(* CODESYS project SmartTraffic.project

Project tree, tasks and I/O mapping:
  Device : CODESYS Control Win V3, 3S - Smart Software Solutions GmbH, order no. 305021, version 3.5.5.50
    application Application
      libraries: Standard, * (System); MQTT Client Library, 3.5.13.20 (Stefan Roßmann Engineering Solutions)
      task MainTask (cyclic, interval t#20ms, priority 1) calls PLC_PRG
      task VISU_TASK (cyclic, interval 100 ms, priority 31) calls VisuElems.Visu_Prg
      program PLC_PRG [CFC]
      function block TrafficLight [ST]
      visualisation Visualization
  text list GlobalTextList
*)

// Device/Application/PLC_PRG
PROGRAM PLC_PRG
VAR
	MQTT_Client_FB_MQTTClient_1 : MQTT_Client.FB_MQTTClient;
	TrafficLight_1: TrafficLight;
END_VAR

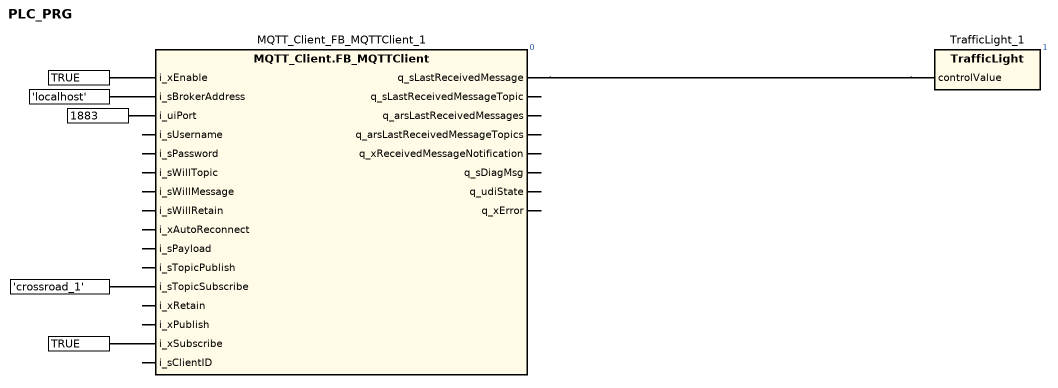
MQTT_Client_FB_MQTTClient_1(
    i_xEnable := TRUE,
    i_sBrokerAddress := 'localhost',
    i_uiPort := 1883,
    i_sTopicSubscribe := 'crossroad_1',
    i_xSubscribe := TRUE); // MQTT_Client.FB_MQTTClient
TrafficLight_1(controlValue := MQTT_Client_FB_MQTTClient_1.q_sLastReceivedMessage); // TrafficLight

END_PROGRAM

// Device/Application/TrafficLight
FUNCTION_BLOCK TrafficLight
VAR_INPUT
	controlValue: STRING;
END_VAR
VAR_OUTPUT
END_VAR
VAR
	Street1Red:BOOL;
	Street1Green:BOOL;
	Street2Red:BOOL;
	Street2Green:BOOL;
	Amber:BOOL;
	Street_TON_1:TON;
	Street_TON_2:TON;
	controlValue_TON_3:TON;
	lastControlValue: STRING;
	street1: TIME := T#15S;
	street2: TIME := T#15S;
	CTU_1: CTU;
	R_TRIG_1: R_TRIG;
END_VAR

CTU_1(PV:= 1, CU:= controlValue_TON_3.Q);
IF CTU_1.Q THEN 
	IF controlValue = 'Increase' THEN 
		street1:= street1 + T#10S;
		street2:= street2 - T#10S;
	ELSIF controlValue = 'Lower' THEN 
		street1:= street1 - T#10S;
		street2:= street2 + T#10S;
	END_IF
	CTU_1(RESET:= TRUE);
	CTU_1(RESET:= FALSE);
	controlValue_TON_3(IN :=FALSE);
END_IF
controlValue_TON_3(IN := TRUE, PT := T#15S);
street1:= LIMIT(T#15S, street1, T#120S);
street2:= LIMIT(T#15S, street2, T#120S);
Street_TON_1(IN := NOT Street_TON_2.Q, PT := street1);
Street_TON_2(IN := Street_TON_1.Q, PT := street2);
Street1Red := Street_TON_1.IN AND NOT Street_TON_1.Q;
Street2Red := Street_TON_1.Q;
Street1Green := NOT Street1Red;
Street2Green := NOT Street2Red;
Amber :=( Street_TON_1.PT - Street_TON_1.ET <= T#3S AND NOT Street_TON_1.Q ) OR Street_TON_2.PT - Street_TON_2.ET <= T#3S;

END_FUNCTION_BLOCK

// Device/Application/Visualization
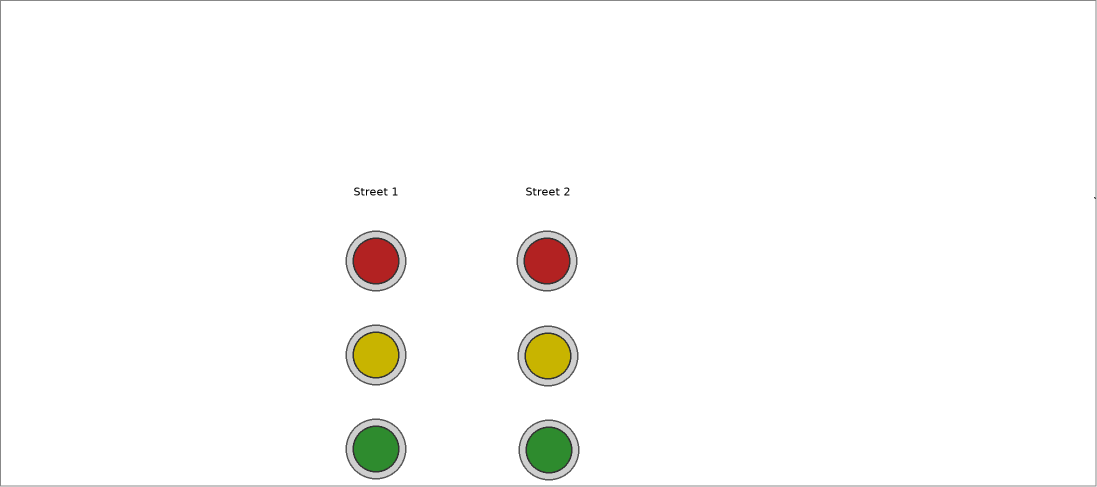
VISUALIZATION Visualization  // 1097x487
    Lamp1 (341,320 70x70), variable: PLC_PRG.TrafficLight_1.Amber, style: Lamp-Lamp1-Yellow
    Polygon (1094,197) (1095,198)
    Label (301,177 150x30), "Street 1"
    Label (473,177 150x30), "Street 2"
    Lamp1 (341,226 70x70), variable: PLC_PRG.TrafficLight_1.Street1Red, style: Lamp-Lamp1-Red
    Lamp1 (341,414 70x70), variable: PLC_PRG.TrafficLight_1.Street1Green, style: Lamp-Lamp1-Green
    Lamp1 (514,415 70x70), variable: PLC_PRG.TrafficLight_1.Street2Green, style: Lamp-Lamp1-Green
    Lamp1 (513,321 70x70), variable: PLC_PRG.TrafficLight_1.Amber, style: Lamp-Lamp1-Yellow
    Lamp1 (512,226 70x70), variable: PLC_PRG.TrafficLight_1.Street2Red, style: Lamp-Lamp1-Red
END_VISUALIZATION
